INTERFACE I_BoolResultTask EXTENDS I_Task

PROPERTY Result : BOOL
GET
END_GET
END_PROPERTY

END_INTERFACE

(* stored: Version 1.1.0.1
   Itf I_BoolResultTask: Id {d224594f-8b3b-4c58-9de9-361ffc3f2952}
   Property Result: Id {d5d593cd-8172-4dc2-86fd-10caaca73c1c}
   Get Get: Id {11a9f9a2-afd6-4d7f-8c9a-c7d3670e9b7f} *)
